// TIA Portal V16 export
// export: Created 2021-05-25T16:14:30.9918315Z, ExportSetting WithDefaults, DisplayName Totally Integrated Automation Portal, DisplayVersion V16, DisplayName TIA Portal Version Control Interface, DisplayVersion V16, DisplayName TIA Portal Openness, DisplayVersion V16, DisplayName STEP 7 Professional, DisplayVersion V16, DisplayName STEP 7 Safety, DisplayVersion V16, DisplayName WinCC Unified SCADA Engineering System, DisplayVersion V16
ORGANIZATION_BLOCK "Profile"   // OB57, LAD, Profile
TITLE = "DP:manufacture_alarm"
{ S7_Optimized_Access := 'TRUE' }
VERSION : 0.1
// stored: IsIECCheckEnabled false, SetENOAutomatically false
   VAR_INPUT
      LADDR : HW_IO;   // Hardware identifier
      Slot : UInt;   // Slot number
      Specifier : Word;   // alarm specifier out of the alarm telegram
   END_VAR
BEGIN
END_ORGANIZATION_BLOCK
